PROGRAM Z_INTRO
VAR
END_VAR

(*-------------------------------------------------------------------------------------------------------*)
(*v050  Introducción Rápida*)
Mc._12_INTRO.v050_Fast.xOpen:= F_INTRO_TK2.z_IntroFast OR
								F_RECIRCULA_TK2.z_TransferTK;

(*-------------------------------------------------------------------------------------------------------*)
(*v051  Introducción Lenta*)
Mc._12_INTRO.v051_Slow.xOpen:= F_INTRO_TK2.z_IntroSlow;

(*-------------------------------------------------------------------------------------------------------*)
(*v055  Modulanta Introducción*)

END_PROGRAM

(* stored: Version 1.1.0.1, ProductVersion 3.1.4024.10
   POU Z_INTRO: Id {85262cb9-f554-487b-9ab9-930e9a314746}, SpecialFunc None *)
